(* PLC project KinIn_v3.project, CODESYS CODESYS V3.5 SP19 *)
(* stored: creationDateTime 2025-01-20T16:27:42.9712604, modificationDateTime 2025-01-20T16:17:39.6822999 *)

FUNCTION_BLOCK Trace
  VAR_INPUT
    {attribute 'variable_length_array_original_scope' := 'Inout'}
    {attribute 'variable_length_array' := 'ARRAY[*,*] OF REAL'}
    {attribute 'Dimensions' := '2'}
    Matrix : POINTER TO REAL;
  END_VAR
  VAR_OUTPUT
    trace : REAL;
  END_VAR
  VAR
    i : DINT;
    j : DINT;
  END_VAR

            trace:=0;
FOR i:=1 TO UPPER_BOUND(Matrix,1) DO
	FOR j:=1 TO UPPER_BOUND(Matrix,2) DO
		IF (i=j) THEN
			trace:=trace+Matrix[i,j];
		END_IF
	END_FOR
END_FOR
          
END_FUNCTION_BLOCK
